Universal Robots PolyScope program: bearing_plate_positioning.urp

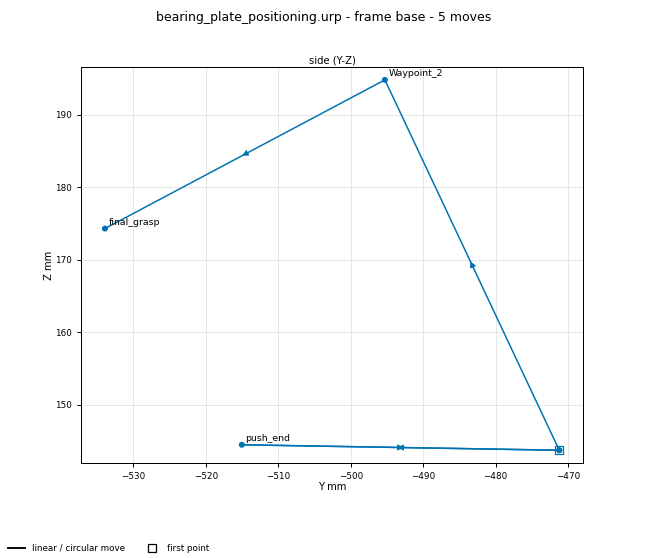
[picture p0: tool path of bearing_plate_positioning.urp in frame base, 5 of 6 moves have a stored position in this frame; points joined in program order, loops and branches not executed]
Program bearing_plate_positioning (installation=default directory=/programs/wrs2020 createdIn=5.9.1.1031110 lastSavedIn=5.9.1.1031110 robotSerialNumber=20205500180)
Calibrated DH parameters: a=[0, -0.425, -0.3922, 0, 0, 0]; d=[0.1625, 0, 0, 0.1333, 0.0997, 0.0996]; alpha=[1.570796, 0, 0, 1.570796, -1.570796, 0]; deltaTheta=[0, 0, 0, 0, 0, 0]
Robot Program (runOnlyOnce=true)
  MoveJ speed 60 deg/s, acceleration 80 deg/s^2 (useActiveTCP=true) feature=Base
    currentpose := get_actual_tcp_pose()get_actual_joint_positions()
    Waypoint Waypoint (Variable): variable=currentpose
  MoveL speed 250 mm/s, acceleration 1200 mm/s^2 (useActiveTCP=false) tcp=gripper_140_tip; feature=Base
    Waypoint before_push: TCP in base x=89.226 y=-471.213 z=143.721 mm, rx=0.0041 ry=3.141 rz=0.0085 rad; joints [84.58, -91.284, 109.644, -108.049, -89.993, -5.272] deg; TCP offset x=0 y=0 z=220 mm, rx=0 ry=0 rz=0 rad
  URCap Gripper (Robotiq_Grippers, Robotiq Inc.) dataModel(position=100.0, force=0.0, speed=0.0, positionInDouble=100.0, forceInDouble=0.0, speedInDouble=0.0, slaveIds=[9], blocking=true)
  MoveL speed 250 mm/s, acceleration 1200 mm/s^2 (useActiveTCP=false) tcp=gripper_140_tip; feature=Base
    Waypoint push_end: motionParameters(jointSpeed=1.047198 jointAcceleration=1.396263 cartesianSpeed=0.02 cartesianAcceleration=0.01); TCP in base x=89.23 y=-515.032 z=144.477 mm, rx=0.0039 ry=3.1409 rz=-0.029 rad; joints [84.975, -86.257, 104.749, -109.542, -89.874, -4.881] deg; TCP offset x=0 y=0 z=220 mm, rx=0 ry=0 rz=0 rad
    Waypoint before_push: motionParameters(jointSpeed=1.047198 jointAcceleration=1.396263 cartesianSpeed=0.25 cartesianAcceleration=0.5); TCP in base x=89.226 y=-471.213 z=143.721 mm, rx=0.0041 ry=3.141 rz=0.0085 rad; joints [84.58, -91.284, 109.644, -108.049, -89.993, -5.272] deg; TCP offset x=0 y=0 z=220 mm, rx=0 ry=0 rz=0 rad
  URCap Gripper (Robotiq_Grippers, Robotiq Inc.) dataModel(position=0.0, force=100.0, speed=100.0, positionInDouble=0.0, forceInDouble=100.0, speedInDouble=100.0, slaveIds=[9], blocking=true)
  MoveL speed 250 mm/s, acceleration 1200 mm/s^2 (useActiveTCP=false) tcp=gripper_140_tip; feature=Base
    Waypoint Waypoint_2: TCP in base x=89.229 y=-495.285 z=194.846 mm, rx=0.0168 ry=3.034 rz=-0.7765 rad; joints [82.081, -107.449, 128.407, -139.394, -85.816, -6.224] deg
    Waypoint final_grasp: TCP in base x=89.247 y=-533.927 z=174.318 mm, rx=0.0137 ry=2.8434 rz=-1.3083 rad; joints [80.631, -99.839, 144.21, -183.366, -82.507, -5.398] deg
  URCap Gripper (Robotiq_Grippers, Robotiq Inc.) dataModel(position=100.0, force=0.0, speed=0.0, positionInDouble=100.0, forceInDouble=0.0, speedInDouble=0.0, slaveIds=[9], blocking=true)
  URCap Gripper (Robotiq_Grippers, Robotiq Inc.) dataModel(position=82.3529411764706, force=100.0, speed=0.0, positionInDouble=82.3529411764706, forceInDouble=100.0, speedInDouble=0.0, slaveIds=[9], blocking=true)
